TYPE ST_P_BARCODE_READ :
STRUCT
	IpAddress:					STRING;
	Port:						STRING;
	Start:						STRING;
	End:						STRING;
	Error:						STRING;
	Barcode:					INT;
END_STRUCT
END_TYPE

(* stored: Version 1.1.0.1, ProductVersion 3.1.4024.10
   DUT ST_P_BARCODE_READ: Id {44a17c0d-e44e-4f30-acd4-ac96594465c2} *)
